FUNCTION_BLOCK Performance5 (* Composite Function Block Type *)
  (* Standard: 61499-2 *)
  (* Version 1.0, 2020-12-26, jetbrains *)
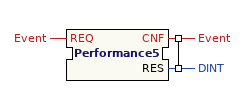
  EVENT_INPUT
    REQ; (* Normal Execution Request *)
  END_EVENT
  EVENT_OUTPUT
    CNF WITH RES; (* Execution Confirmation *)
  END_EVENT
  VAR_OUTPUT
    RES : DINT; (* Output event qualifier *)
  END_VAR
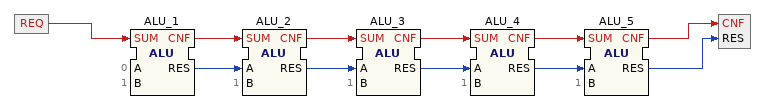
  FBS
    ALU_1 : ALU(A := 0, B := 1);
    ALU_2 : ALU(B := 1);
    ALU_3 : ALU(B := 1);
    ALU_4 : ALU(B := 1);
    ALU_5 : ALU(B := 1);
  END_FBS
  EVENT_CONNECTIONS
    ALU_1.CNF TO ALU_2.SUM;
    ALU_2.CNF TO ALU_3.SUM;
    ALU_4.CNF TO ALU_5.SUM;
    ALU_3.CNF TO ALU_4.SUM;
    REQ TO ALU_1.SUM;
    ALU_5.CNF TO CNF;
  END_CONNECTIONS
  DATA_CONNECTIONS
    ALU_1.RES TO ALU_2.A;
    ALU_4.RES TO ALU_5.A;
    ALU_3.RES TO ALU_4.A;
    ALU_2.RES TO ALU_3.A;
    ALU_5.RES TO RES;
  END_CONNECTIONS
END_FUNCTION_BLOCK
